INTERFACE ILine EXTENDS IStringContainer

METHOD splitBy : IStringContainerList
VAR_INPUT
	splitter	: STRING(255);
	addEmptyEntries :BOOL := FALSE;
END_VAR
END_METHOD

END_INTERFACE

(* stored: Version 1.1.0.1
   Itf ILine: Id {f12f8a50-77ce-4b32-8977-4d350efde387}
   Method splitBy: Id {c7d5a0a2-a8b4-4157-82a2-6f0ab10f5ea6} *)
